FUNCTION_BLOCK FB_Connection EXTENDS FB_Basis
VAR_INPUT
	IP						:STRING(MAX_STRING_LENGTH);
	NameSpace				:STRING(MAX_STRING_LENGTH);
END_VAR

VAR_OUTPUT
	NodeHdl_SW				:DWORD;
	NodeHdl_CW				:DWORD;	
END_VAR

VAR
	// Instanziierung der Kommunikationsfunktionsblöcke
	Connect					:UA_Connect;
	NameSpaceInd			:UA_GetNamespaceIndex;
	Node_SW					:UA_NodeGetHandle;
	Node_CW					:UA_NodeGetHandle;
	
	// Instanziierung der relevanten Input-Variablen
	ConnectInfo				:ST_UASessionConnectInfo;			// Informationen für Verbindungsaufbau 
	NodeID_SW				:ST_UANodeID;
	NodeID_CW				:ST_UANodeID;
	NodeIdentifier_SW		:STRING(MAX_STRING_LENGTH) := 'GVL_OPC_UA.SW';
	NodeIdentifier_CW		:STRING(MAX_STRING_LENGTH) := 'GVL_OPC_UA.CW';
	
	// Instanziierung der relevanten Output-Variablen
	ConnectionHdl			:DWORD;								// Connection-Handle
	NameSpaceIndex			:UINT;
END_VAR

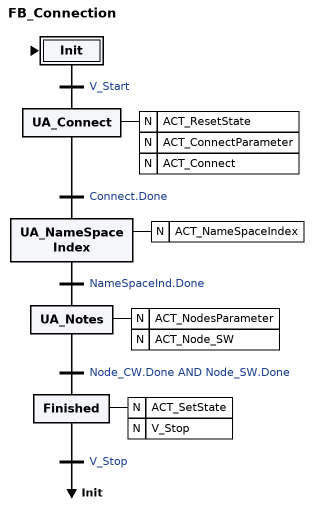
INITIAL_STEP Init:
END_STEP
TRANSITION FROM Init TO UA_Connect
    := V_Start;
END_TRANSITION
STEP UA_Connect:
    ACT_ResetState(N);
    ACT_ConnectParameter(N);
    ACT_Connect(N);
END_STEP
TRANSITION FROM UA_Connect TO UA_NameSpaceIndex
    := Connect.Done;
END_TRANSITION
STEP UA_NameSpaceIndex:
    ACT_NameSpaceIndex(N);
END_STEP
TRANSITION FROM UA_NameSpaceIndex TO UA_Notes
    := NameSpaceInd.Done;
END_TRANSITION
STEP UA_Notes:
    ACT_NodesParameter(N);
    ACT_Node_SW(N);
END_STEP
TRANSITION FROM UA_Notes TO Finished
    := Node_CW.Done AND Node_SW.Done;
END_TRANSITION
STEP Finished:
    ACT_SetState(N);
    V_Stop(N);
END_STEP
TRANSITION FROM Finished TO Init
    := V_Stop;
END_TRANSITION

ACTION ACT_Connect:
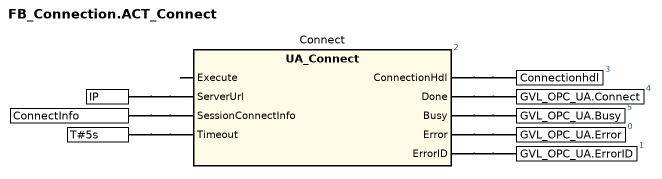
GVL_OPC_UA.Error := Connect.Error;
GVL_OPC_UA.ErrorID := Connect.ErrorID;
Connect(ServerUrl := IP, SessionConnectInfo := ConnectInfo, Timeout := T#5s); // UA_Connect
Connectionhdl := Connect.ConnectionHdl;
GVL_OPC_UA.Connect := Connect.Done;
GVL_OPC_UA.Busy := Connect.Busy;
END_ACTION

ACTION ACT_ConnectParameter:
// Definition der Verbindungsinformationen
ConnectInfo.tSessionTimeout := T#1M;
ConnectInfo.tConnectTimeout := T#1M;
ConnectInfo.sApplicationName := '';
ConnectInfo.eSecurityMode := eUASecurityMsgMode_Sign_Encrypt;				// 3 = Sign_Encrypted
ConnectInfo.eSecurityPolicyUri := eUASecurityPolicy_Basic256Sha256;			// 4 = Basic256  
ConnectInfo.eTransportProfileUri := eUATransportProfileUri_UATcp;			// 1 = UATcp
ConnectInfo.stUserIdentTokenType.eUserIdentTokenType := eUAUITT_Username;	// 1 = Username
ConnectInfo.stUserIdentTokenType.sTokenParam1 := 'Administrator';			// Username
ConnectInfo.stUserIdentTokenType.sTokenParam2 := '1';						// PW

Connect.Execute := TRUE;
NameSpaceInd.Execute := TRUE;
END_ACTION

ACTION ACT_NameSpaceIndex:
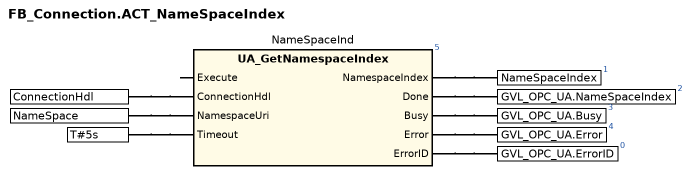
GVL_OPC_UA.ErrorID := NameSpaceInd.ErrorID;
NameSpaceIndex := NameSpaceInd.NamespaceIndex;
GVL_OPC_UA.NameSpaceIndex := NameSpaceInd.Done;
GVL_OPC_UA.Busy := NameSpaceInd.Busy;
GVL_OPC_UA.Error := NameSpaceInd.Error;
NameSpaceInd(ConnectionHdl := ConnectionHdl, NamespaceUri := NameSpace, Timeout := T#5s); // UA_GetNamespaceIndex
END_ACTION

ACTION ACT_Node_CW:
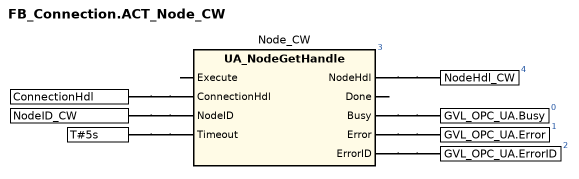
GVL_OPC_UA.Busy := Node_CW.Busy;
GVL_OPC_UA.Error := Node_CW.Error;
GVL_OPC_UA.ErrorID := Node_CW.ErrorID;
Node_CW(ConnectionHdl := ConnectionHdl, NodeID := NodeID_CW, Timeout := T#5s); // UA_NodeGetHandle
NodeHdl_CW := Node_CW.NodeHdl;
END_ACTION

ACTION ACT_Node_SW:
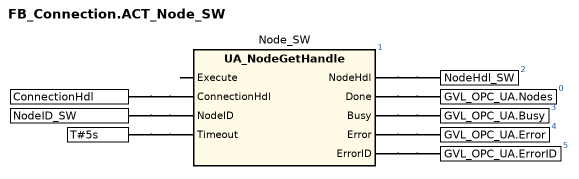
GVL_OPC_UA.Nodes := Node_SW.Done;
Node_SW(ConnectionHdl := ConnectionHdl, NodeID := NodeID_SW, Timeout := T#5s); // UA_NodeGetHandle
NodeHdl_SW := Node_SW.NodeHdl;
GVL_OPC_UA.Busy := Node_SW.Busy;
GVL_OPC_UA.Error := Node_SW.Error;
GVL_OPC_UA.ErrorID := Node_SW.ErrorID;
END_ACTION

ACTION ACT_NodesParameter:
// Definieren von relevanten Parameter

// Statusword - SW
NodeID_SW.eIdentifierType := eUAIdentifierType_String;
NodeID_SW.nNamespaceIndex := NameSpaceIndex;
NodeID_SW.sIdentifier := NodeIdentifier_SW;

// Controlword - CW
NodeID_CW.eIdentifierType := eUAIdentifierType_String;
NodeID_CW.nNamespaceIndex := NameSpaceIndex;
NodeID_CW.sIdentifier := NodeIdentifier_CW;

Node_CW.Execute := TRUE;
Node_SW.Execute := TRUE;
END_ACTION

ACTION ACT_ResetState:
GVL.ConnectionState := 0;
END_ACTION

ACTION ACT_SetState:
GVL.ConnectionState := 1;
END_ACTION

END_FUNCTION_BLOCK

(* stored: Version 1.1.0.1, ProductVersion 3.1.4024.12
   POU FB_Connection: Id {cd7cf23f-492d-4c5e-b487-83e671b20ca8}, SpecialFunc None
   Folder 01_Aktionen: Id {e0fea88b-373c-4ace-b6f0-b643c89fd156}
   Action ACT_Connect: Id {1715e335-e2a4-4d9f-b49d-70c12bafd1c3}
   Action ACT_ConnectParameter: Id {068bfebf-1546-4ec6-8b8c-9121ed2821a1}
   Action ACT_NameSpaceIndex: Id {57843c14-1fa5-4498-845b-c7a175f21a81}
   Action ACT_Node_CW: Id {0b247d0e-2d01-428a-8405-ab1dfbc182f0}
   Action ACT_Node_SW: Id {6344d690-86b3-4b39-b777-c24a36170fed}
   Action ACT_NodesParameter: Id {f77fda67-af9e-48ac-8f20-50fb6e8efb05}
   Action ACT_ResetState: Id {b2e33ad7-7036-4db1-b566-24d4140e9f24}
   Action ACT_SetState: Id {cce30d94-7e34-4df6-b8e8-b5a539646154} *)
